PROGRAM MAIN
VAR
	bButtonStart,
	bButtonReset,
	bButtonStop: BOOL;
	bStatus : BOOL;
	bButtonLightStart,
	bButtonLightStop,
	bExtra, botroextra,bTercer,bCuarto : BOOL;
END_VAR

bButtonStart := GVL.mb_Output_Coils[0];
bButtonStop := GVL.mb_Output_Coils[1];
bButtonReset := GVL.mb_Output_Coils[29];
GVL.mb_Input_Coils[0] := bButtonLightStart;
GVL.mb_Input_Coils[1] := bButtonLightStop;
conveyor1();

Tags.bAutoMan(SET1 := bButtonStart, RESET := NOT bButtonStop);
bStatus := Tags.bAutoMan.Q1;
bButtonLightStart := bStatus;
bButtonLightStop := not bStatus;

END_PROGRAM

(* stored: Version 1.1.0.1, ProductVersion 3.1.4024.12
   POU MAIN: Id {a7fd1c1b-457e-4c34-afce-02d523ac5831}, SpecialFunc None *)
